// TIA Portal V20 export
TYPE "LER_typeVisionTrackingData"
// stored: Access Published
   STRUCT
      finished { ExternalWritable := 'False'} : Bool;
      result { ExternalWritable := 'False'} : Bool;
      data0 { ExternalWritable := 'False'} : Array[0..15] of Byte;
      data1 { ExternalWritable := 'False'} : Array[0..31] of Byte;
      data2 { ExternalWritable := 'False'} : Array[0..31] of Byte;
      data3 { ExternalWritable := 'False'} : Array[0..31] of Byte;
      data4 { ExternalWritable := 'False'} : Array[0..31] of Byte;
      data5 { ExternalWritable := 'False'} : Array[0..31] of Byte;
   END_STRUCT;
END_TYPE
